Fanuc KAREL source: kb00117.KL

-- PROVISIONAL review KL for V770-1; original PC SHA256 c2453351cc948074077e86c996a230ee93b94b5d3e50b8d3eb6bd2ca3d1f4576
-- Incomplete behavior may be omitted. Consult companion uncertainty JSON. Do not deploy.
PROGRAM KB00117
%NOLOCKGROUP
BEGIN
  -- UNRESOLVED_PC offsets 5-14; opcodes 3F,75
  -- UNRESOLVED_PC offsets 19-26; opcodes 9D,23
  -- UNRESOLVED_PC offsets 31-38; opcodes 9D,23
  -- UNRESOLVED_PC offsets 43-67; opcodes 27,22,2A,22,22,31
  -- UNRESOLVED_PC offsets 72-76; opcodes 7F
END KB00117
